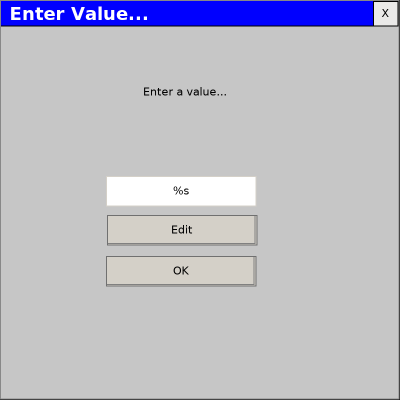
VISUALIZATION dialogEnterValue  // 400x400
VAR_IN_OUT
	enteredValue:string;
	
END_VAR
    Rectangle (0,0 400x400)
    Rectangle (0,0 400x26), "Enter Value..."
    Rectangle (373,1 25x25), "X"
        OnMouseClick: CloseDialog Dialog=dialogEnterValue, Result=Cancel, NumpadKeypadSet=True
    Label (110,77 150x30), "Enter a value..."
    Textfield (106,176 150x30), "%s", text variable: enteredValue
    Button (107,215 150x30), "Edit"
        OnMouseClick: write enteredValue via VisuDialogs.Numpad
    Button (106,256 150x30), "OK"
        OnMouseClick: CloseDialog Dialog=dialogEnterValue, Result=OK, NumpadKeypadSet=True
END_VISUALIZATION

(* stored: Version 1.1.0.1, ProductVersion 3.1.4024.11
   Visu dialogEnterValue: Id {f98eb1f3-4b2f-0a4f-0a42-60ac8083e0aa} *)
